LIN {X 0,Y 123.442,Z 476.669,A -85,B 0,C 180,E1 -28629.835,E2 -28629.835} C_VEL
LIN {X 0,Y 123.131,Z 478.566,A -85,B 0,C 180,E1 -28633.994,E2 -28633.994} C_VEL
LIN {X 0,Y 122.926,Z 480.125,A -85,B 0,C 180,E1 -28636.611,E2 -28636.611} C_VEL
LIN {X 0,Y 122.223,Z 482.877,A -85,B 0,C 180,E1 -28640.183,E2 -28640.183} C_VEL
LIN {X 0,Y 121.163,Z 486.4,A -85,B 0,C 180,E1 -28643.956,E2 -28643.956} C_VEL
LIN {X 0,Y 120.084,Z 488.681,A -85,B 0,C 180,E1 -28645.839,E2 -28645.839} C_VEL
LIN {X 0,Y 110.646,Z 498.011,A -85,B 0,C 180,E1 -28649.147,E2 -28649.147} C_VEL
LIN {X 0,Y 100.856,Z 506.281,A -85,B 0,C 180,E1 -28653.259,E2 -28653.259} C_VEL
LIN {X 0,Y 92.106,Z 512.776,A -85,B 0,C 180,E1 -28658.074,E2 -28658.074} C_VEL
LIN {X 0,Y 83.54,Z 518.436,A -85,B 0,C 180,E1 -28664.35,E2 -28664.35} C_VEL
LIN {X 0,Y 75.32,Z 523.224,A -85,B 0,C 180,E1 -28672.663,E2 -28672.663} C_VEL
LIN {X 0,Y 68.671,Z 526.759,A -85,B 0,C 180,E1 -28683.323,E2 -28683.323} C_VEL
LIN {X 0,Y 66.155,Z 527.832,A -85,B 0,C 180,E1 -28687.77,E2 -28687.77} C_VEL
LIN {X 0,Y 61.137,Z 529.24,A -85,B 0,C 180,E1 -28695.36,E2 -28695.36} C_VEL
LIN {X 0,Y 57.636,Z 529.91,A -85,B 0,C 180,E1 -28702.265,E2 -28702.265} C_VEL
LIN {X 0,Y 56.173,Z 530.076,A -85,B 0,C 180,E1 -28708.082,E2 -28708.082} C_VEL
LIN {X 0,Y 56.026,Z 530.057,A -85,B 0,C 180,E1 -28710.105,E2 -28710.105} C_VEL
LIN {X 0,Y 57.314,Z 529.481,A -85,B 0,C 180,E1 -28724.197,E2 -28724.197} C_VEL
LIN {X 0,Y 61.277,Z 527.703,A -85,B 0,C 180,E1 -28737.309,E2 -28737.309} C_VEL
LIN {X 0,Y 67.813,Z 524.66,A -85,B 0,C 180,E1 -28748.451,E2 -28748.451} C_VEL
LIN {X 0,Y 73.975,Z 521.492,A -85,B 0,C 180,E1 -28755.443,E2 -28755.443} C_VEL
LIN {X 0,Y 83.706,Z 515.997,A -85,B 0,C 180,E1 -28762.905,E2 -28762.905} C_VEL
LIN {X 0,Y 91.522,Z 510.885,A -85,B 0,C 180,E1 -28767.641,E2 -28767.641} C_VEL
LIN {X 0,Y 101.389,Z 503.57,A -85,B 0,C 180,E1 -28772.105,E2 -28772.105} C_VEL
LIN {X 0,Y 111.81,Z 494.625,A -85,B 0,C 180,E1 -28775.704,E2 -28775.704} C_VEL
LIN {X 0,Y 114.82,Z 491.688,A -85,B 0,C 180,E1 -28776.656,E2 -28776.656} C_VEL
LIN {X 0,Y 115.99,Z 490.149,A -85,B 0,C 180,E1 -28777.717,E2 -28777.717} C_VEL
LIN {X 0,Y 117.045,Z 487.526,A -85,B 0,C 180,E1 -28780.715,E2 -28780.715} C_VEL
LIN {X 0,Y 117.659,Z 485.914,A -85,B 0,C 180,E1 -28782.887,E2 -28782.887} C_VEL
LIN {X 0,Y 118.148,Z 483.965,A -85,B 0,C 180,E1 -28786.234,E2 -28786.234} C_VEL
LIN {X 0,Y 118.549,Z 482.415,A -85,B 0,C 180,E1 -28789.755,E2 -28789.755} C_VEL
LIN {X 0,Y 118.914,Z 481.354,A -85,B 0,C 180,E1 -28793.211,E2 -28793.211} C_VEL
LIN {X 0,Y 119.159,Z 480.799,A -85,B 0,C 180,E1 -28796.618,E2 -28796.618} C_VEL
LIN {X 0,Y 119.149,Z 480.971,A -85,B 0,C 180,E1 -28799.999,E2 -28799.999} C_VEL
LIN {X 0,Y 118.814,Z 481.957,A -85,B 0,C 180,E1 -28803.39,E2 -28803.39} C_VEL
LIN {X 0,Y 118.391,Z 483.416,A -85,B 0,C 180,E1 -28806.818,E2 -28806.818} C_VEL
LIN {X 0,Y 117.865,Z 485.41,A -85,B 0,C 180,E1 -28810.304,E2 -28810.304} C_VEL
LIN {X 0,Y 117.082,Z 488.121,A -85,B 0,C 180,E1 -28813.892,E2 -28813.892} C_VEL
LIN {X 0,Y 115.532,Z 492.582,A -85,B 0,C 180,E1 -28818.794,E2 -28818.794} C_VEL
LIN {X 0,Y 115.01,Z 493.547,A -85,B 0,C 180,E1 -28819.533,E2 -28819.533} C_VEL
LIN {X 0,Y 104.738,Z 503.117,A -85,B 0,C 180,E1 -28822.683,E2 -28822.683} C_VEL
LIN {X 0,Y 94.468,Z 511.413,A -85,B 0,C 180,E1 -28826.778,E2 -28826.778} C_VEL
LIN {X 0,Y 83.489,Z 519.074,A -85,B 0,C 180,E1 -28832.669,E2 -28832.669} C_VEL
LIN {X 0,Y 73.567,Z 525.093,A -85,B 0,C 180,E1 -28840.158,E2 -28840.158} C_VEL
LIN {X 0,Y 65.334,Z 529.662,A -85,B 0,C 180,E1 -28849.801,E2 -28849.801} C_VEL
LIN {X 0,Y 59.215,Z 532.878,A -85,B 0,C 180,E1 -28861.656,E2 -28861.656} C_VEL
LIN {X 0,Y 55.998,Z 534.817,A -85,B 0,C 180,E1 -28875.462,E2 -28875.462} C_VEL
LIN {X 0,Y 55.744,Z 535.501,A -85,B 0,C 180,E1 -28889.999,E2 -28889.999} C_VEL
LIN {X 0,Y 55.999,Z 534.796,A -85,B 0,C 180,E1 -28904.536,E2 -28904.536} C_VEL
LIN {X 0,Y 59.195,Z 532.826,A -85,B 0,C 180,E1 -28918.353,E2 -28918.353} C_VEL
LIN {X 0,Y 65.247,Z 529.584,A -85,B 0,C 180,E1 -28930.261,E2 -28930.261} C_VEL
LIN {X 0,Y 73.545,Z 524.995,A -85,B 0,C 180,E1 -28939.861,E2 -28939.861} C_VEL
LIN {X 0,Y 83.473,Z 518.938,A -85,B 0,C 180,E1 -28947.347,E2 -28947.347} C_VEL
LIN {X 0,Y 94.427,Z 511.231,A -85,B 0,C 180,E1 -28953.27,E2 -28953.27} C_VEL
LIN {X 0,Y 104.716,Z 502.903,A -85,B 0,C 180,E1 -28957.344,E2 -28957.344} C_VEL
LIN {X 0,Y 114.943,Z 493.322,A -85,B 0,C 180,E1 -28960.492,E2 -28960.492} C_VEL
LIN {X 0,Y 115.872,Z 491.229,A -85,B 0,C 180,E1 -28962.347,E2 -28962.347} C_VEL
LIN {X 0,Y 117.35,Z 486.686,A -85,B 0,C 180,E1 -28967.619,E2 -28967.619} C_VEL
LIN {X 0,Y 117.773,Z 485.194,A -85,B 0,C 180,E1 -28969.688,E2 -28969.688} C_VEL
LIN {X 0,Y 118.264,Z 483.229,A -85,B 0,C 180,E1 -28973.175,E2 -28973.175} C_VEL
LIN {X 0,Y 118.678,Z 481.763,A -85,B 0,C 180,E1 -28976.606,E2 -28976.606} C_VEL
LIN {X 0,Y 119.054,Z 480.719,A -85,B 0,C 180,E1 -28980.001,E2 -28980.001} C_VEL
LIN {X 0,Y 119.069,Z 480.536,A -85,B 0,C 180,E1 -28983.384,E2 -28983.384} C_VEL
LIN {X 0,Y 118.726,Z 481.294,A -85,B 0,C 180,E1 -28987.438,E2 -28987.438} C_VEL
LIN {X 0,Y 118.472,Z 482.151,A -85,B 0,C 180,E1 -28990.252,E2 -28990.252} C_VEL
LIN {X 0,Y 118.083,Z 483.683,A -85,B 0,C 180,E1 -28993.773,E2 -28993.773} C_VEL
LIN {X 0,Y 117.525,Z 485.84,A -85,B 0,C 180,E1 -28997.398,E2 -28997.398} C_VEL
LIN {X 0,Y 115.975,Z 489.809,A -85,B 0,C 180,E1 -29002.234,E2 -29002.234} C_VEL
LIN {X 0,Y 114.863,Z 491.379,A -85,B 0,C 180,E1 -29003.395,E2 -29003.395} C_VEL
LIN {X 0,Y 104.387,Z 500.893,A -85,B 0,C 180,E1 -29006.864,E2 -29006.864} C_VEL
LIN {X 0,Y 94.332,Z 508.689,A -85,B 0,C 180,E1 -29011.043,E2 -29011.043} C_VEL
LIN {X 0,Y 86.254,Z 514.244,A -85,B 0,C 180,E1 -29015.432,E2 -29015.432} C_VEL
LIN {X 0,Y 78.74,Z 518.785,A -85,B 0,C 180,E1 -29020.653,E2 -29020.653} C_VEL
LIN {X 0,Y 69.786,Z 523.572,A -85,B 0,C 180,E1 -29029.111,E2 -29029.111} C_VEL
LIN {X 0,Y 62.167,Z 527.216,A -85,B 0,C 180,E1 -29040.869,E2 -29040.869} C_VEL
LIN {X 0,Y 58.97,Z 528.699,A -85,B 0,C 180,E1 -29049.052,E2 -29049.052} C_VEL
LIN {X 0,Y 56.296,Z 529.907,A -85,B 0,C 180,E1 -29062.829,E2 -29062.829} C_VEL
LIN {X 0,Y 56.026,Z 530.057,A -85,B 0,C 180,E1 -29070.105,E2 -29070.105} C_VEL
LIN {X 0,Y 55.496,Z 529.985,A -85,B 0,C 180,E1 -29076.152,E2 -29076.152} C_VEL
LIN {X 0,Y 54.053,Z 529.556,A -85,B 0,C 180,E1 -29086.427,E2 -29086.427} C_VEL
LIN {X 0,Y 53.917,Z 528.842,A -85,B 0,C 180,E1 -29094.874,E2 -29094.874} C_VEL
LIN {X 0,Y 55.248,Z 528.005,A -85,B 0,C 180,E1 -29100.892,E2 -29100.892} C_VEL
LIN {X 0,Y 56.05,Z 527.625,A -85,B 0,C 180,E1 -29102.721,E2 -29102.721} C_VEL
LIN {X 0,Y 64.524,Z 524.032,A -85,B 0,C 180,E1 -29115.073,E2 -29115.073} C_VEL
LIN {X 0,Y 74.271,Z 519.28,A -85,B 0,C 180,E1 -29123.546,E2 -29123.546} C_VEL
LIN {X 0,Y 84.459,Z 513.418,A -85,B 0,C 180,E1 -29129.824,E2 -29129.824} C_VEL
LIN {X 0,Y 95.251,Z 506.136,A -85,B 0,C 180,E1 -29134.672,E2 -29134.672} C_VEL
LIN {X 0,Y 105.982,Z 497.686,A -85,B 0,C 180,E1 -29138.187,E2 -29138.187} C_VEL
LIN {X 0,Y 110.875,Z 493.225,A -85,B 0,C 180,E1 -29139.785,E2 -29139.785} C_VEL
LIN {X 0,Y 112.206,Z 490.669,A -85,B 0,C 180,E1 -29143.22,E2 -29143.22} C_VEL
LIN {X 0,Y 112.67,Z 489.356,A -85,B 0,C 180,E1 -29145.551,E2 -29145.551} C_VEL
LIN {X 0,Y 113.3,Z 487.678,A -85,B 0,C 180,E1 -29149.275,E2 -29149.275} C_VEL
LIN {X 0,Y 113.819,Z 486.542,A -85,B 0,C 180,E1 -29152.906,E2 -29152.906} C_VEL
LIN {X 0,Y 114.16,Z 485.933,A -85,B 0,C 180,E1 -29156.47,E2 -29156.47} C_VEL
LIN {X 0,Y 114.154,Z 486.101,A -85,B 0,C 180,E1 -29159.999,E2 -29159.999} C_VEL
LIN {X 0,Y 113.684,Z 487.173,A -85,B 0,C 180,E1 -29163.544,E2 -29163.544} C_VEL
LIN {X 0,Y 113.087,Z 488.722,A -85,B 0,C 180,E1 -29167.139,E2 -29167.139} C_VEL
LIN {X 0,Y 112.312,Z 490.85,A -85,B 0,C 180,E1 -29170.819,E2 -29170.819} C_VEL
LIN {X 0,Y 111.093,Z 493.787,A -85,B 0,C 180,E1 -29174.657,E2 -29174.657} C_VEL
LIN {X 0,Y 110.108,Z 495.718,A -85,B 0,C 180,E1 -29176.776,E2 -29176.776} C_VEL
LIN {X 0,Y 99.067,Z 505.251,A -85,B 0,C 180,E1 -29179.949,E2 -29179.949} C_VEL
LIN {X 0,Y 89.974,Z 512.085,A -85,B 0,C 180,E1 -29183.39,E2 -29183.39} C_VEL
LIN {X 0,Y 79.849,Z 518.722,A -85,B 0,C 180,E1 -29188.336,E2 -29188.336} C_VEL
LIN {X 0,Y 69.139,Z 524.742,A -85,B 0,C 180,E1 -29195.589,E2 -29195.589} C_VEL
LIN {X 0,Y 60.013,Z 529.312,A -85,B 0,C 180,E1 -29205.359,E2 -29205.359} C_VEL
LIN {X 0,Y 53.023,Z 532.53,A -85,B 0,C 180,E1 -29217.981,E2 -29217.981} C_VEL
LIN {X 0,Y 49.106,Z 534.47,A -85,B 0,C 180,E1 -29233.366,E2 -29233.366} C_VEL
LIN {X 0,Y 48.634,Z 535.155,A -85,B 0,C 180,E1 -29249.999,E2 -29249.999} C_VEL
LIN {X 0,Y 49.106,Z 534.448,A -85,B 0,C 180,E1 -29266.632,E2 -29266.632} C_VEL
LIN {X 0,Y 53,Z 532.477,A -85,B 0,C 180,E1 -29282.033,E2 -29282.033} C_VEL
LIN {X 0,Y 59.933,Z 529.232,A -85,B 0,C 180,E1 -29294.715,E2 -29294.715} C_VEL
LIN {X 0,Y 69.125,Z 524.641,A -85,B 0,C 180,E1 -29304.426,E2 -29304.426} C_VEL
LIN {X 0,Y 79.832,Z 518.584,A -85,B 0,C 180,E1 -29311.684,E2 -29311.684} C_VEL
LIN {X 0,Y 91.413,Z 510.868,A -85,B 0,C 180,E1 -29317.306,E2 -29317.306} C_VEL
LIN {X 0,Y 102.167,Z 502.533,A -85,B 0,C 180,E1 -29321.059,E2 -29321.059} C_VEL
LIN {X 0,Y 110.092,Z 495.463,A -85,B 0,C 180,E1 -29323.248,E2 -29323.248} C_VEL
LIN {X 0,Y 111.044,Z 493.576,A -85,B 0,C 180,E1 -29325.336,E2 -29325.336} C_VEL
LIN {X 0,Y 112.232,Z 490.64,A -85,B 0,C 180,E1 -29329.173,E2 -29329.173} C_VEL
LIN {X 0,Y 113.147,Z 488.13,A -85,B 0,C 180,E1 -29333.629,E2 -29333.629} C_VEL
LIN {X 0,Y 113.558,Z 486.983,A -85,B 0,C 180,E1 -29336.452,E2 -29336.452} C_VEL
LIN {X 0,Y 114.055,Z 485.873,A -85,B 0,C 180,E1 -29340.001,E2 -29340.001} C_VEL
LIN {X 0,Y 114.08,Z 485.68,A -85,B 0,C 180,E1 -29343.533,E2 -29343.533} C_VEL
LIN {X 0,Y 113.59,Z 486.589,A -85,B 0,C 180,E1 -29348.132,E2 -29348.132} C_VEL
LIN {X 0,Y 113.231,Z 487.427,A -85,B 0,C 180,E1 -29350.732,E2 -29350.732} C_VEL
LIN {X 0,Y 112.605,Z 489.096,A -85,B 0,C 180,E1 -29354.458,E2 -29354.458} C_VEL
LIN {X 0,Y 112.16,Z 490.362,A -85,B 0,C 180,E1 -29356.693,E2 -29356.693} C_VEL
LIN {X 0,Y 110.825,Z 492.996,A -85,B 0,C 180,E1 -29360.279,E2 -29360.279} C_VEL
LIN {X 0,Y 107.557,Z 496.07,A -85,B 0,C 180,E1 -29361.389,E2 -29361.389} C_VEL
LIN {X 0,Y 96.809,Z 504.795,A -85,B 0,C 180,E1 -29364.844,E2 -29364.844} C_VEL
LIN {X 0,Y 86.811,Z 511.771,A -85,B 0,C 180,E1 -29369.062,E2 -29369.062} C_VEL
LIN {X 0,Y 76.956,Z 517.733,A -85,B 0,C 180,E1 -29374.723,E2 -29374.723} C_VEL
LIN {X 0,Y 66.816,Z 522.882,A -85,B 0,C 180,E1 -29382.584,E2 -29382.584} C_VEL
LIN {X 0,Y 58.485,Z 526.608,A -85,B 0,C 180,E1 -29393.071,E2 -29393.071} C_VEL
LIN {X 0,Y 52.417,Z 529.044,A -85,B 0,C 180,E1 -29406.283,E2 -29406.283} C_VEL
LIN {X 0,Y 49.28,Z 530.252,A -85,B 0,C 180,E1 -29421.802,E2 -29421.802} C_VEL
LIN {X 0,Y 48.949,Z 530.404,A -85,B 0,C 180,E1 -29430.001,E2 -29430.001} C_VEL
LIN {X 0,Y 50.461,Z 529.826,A -85,B 0,C 180,E1 -29446.175,E2 -29446.175} C_VEL
LIN {X 0,Y 55.071,Z 528.048,A -85,B 0,C 180,E1 -29460.696,E2 -29460.696} C_VEL
LIN {X 0,Y 56.05,Z 527.625,A -85,B 0,C 180,E1 -29462.721,E2 -29462.721} C_VEL
LIN {X 0,Y 58.351,Z 526.555,A -85,B 0,C 180,E1 -29468.046,E2 -29468.046} C_VEL
LIN {X 0,Y 61.578,Z 524.441,A -85,B 0,C 180,E1 -29476.786,E2 -29476.786} C_VEL
LIN {X 0,Y 65.945,Z 521.835,A -85,B 0,C 180,E1 -29484.444,E2 -29484.444} C_VEL
LIN {X 0,Y 69.769,Z 519.876,A -85,B 0,C 180,E1 -29487.874,E2 -29487.874} C_VEL
LIN {X 0,Y 78.831,Z 515.114,A -85,B 0,C 180,E1 -29493.067,E2 -29493.067} C_VEL
LIN {X 0,Y 89.345,Z 508.618,A -85,B 0,C 180,E1 -29497.561,E2 -29497.561} C_VEL
LIN {X 0,Y 100.366,Z 500.648,A -85,B 0,C 180,E1 -29500.967,E2 -29500.967} C_VEL
LIN {X 0,Y 106.067,Z 495.905,A -85,B 0,C 180,E1 -29502.611,E2 -29502.611} C_VEL
LIN {X 0,Y 106.883,Z 494.538,A -85,B 0,C 180,E1 -29504.75,E2 -29504.75} C_VEL
LIN {X 0,Y 107.731,Z 492.77,A -85,B 0,C 180,E1 -29508.713,E2 -29508.713} C_VEL
LIN {X 0,Y 108.493,Z 491.5,A -85,B 0,C 180,E1 -29512.555,E2 -29512.555} C_VEL
LIN {X 0,Y 108.936,Z 490.843,A -85,B 0,C 180,E1 -29516.3,E2 -29516.3} C_VEL
LIN {X 0,Y 108.916,Z 491.025,A -85,B 0,C 180,E1 -29519.999,E2 -29519.999} C_VEL
LIN {X 0,Y 108.316,Z 492.16,A -85,B 0,C 180,E1 -29523.72,E2 -29523.72} C_VEL
LIN {X 0,Y 107.558,Z 493.767,A -85,B 0,C 180,E1 -29527.508,E2 -29527.508} C_VEL
LIN {X 0,Y 106.414,Z 496.104,A -85,B 0,C 180,E1 -29531.427,E2 -29531.427} C_VEL
LIN {X 0,Y 104.974,Z 498.293,A -85,B 0,C 180,E1 -29533.882,E2 -29533.882} C_VEL
LIN {X 0,Y 93.645,Z 507.308,A -85,B 0,C 180,E1 -29536.883,E2 -29536.883} C_VEL
LIN {X 0,Y 82.737,Z 514.756,A -85,B 0,C 180,E1 -29540.869,E2 -29540.869} C_VEL
LIN {X 0,Y 70.811,Z 521.57,A -85,B 0,C 180,E1 -29546.713,E2 -29546.713} C_VEL
LIN {X 0,Y 59.957,Z 526.851,A -85,B 0,C 180,E1 -29554.862,E2 -29554.862} C_VEL
LIN {X 0,Y 50.779,Z 530.735,A -85,B 0,C 180,E1 -29566.208,E2 -29566.208} C_VEL
LIN {X 0,Y 44.196,Z 533.307,A -85,B 0,C 180,E1 -29581.506,E2 -29581.506} C_VEL
LIN {X 0,Y 41.413,Z 534.624,A -85,B 0,C 180,E1 -29600.228,E2 -29600.228} C_VEL
LIN {X 0,Y 41.523,Z 534.809,A -85,B 0,C 180,E1 -29609.999,E2 -29609.999} C_VEL
LIN {X 0,Y 42.294,Z 534.099,A -85,B 0,C 180,E1 -29629.41,E2 -29629.41} C_VEL
LIN {X 0,Y 47.059,Z 532.127,A -85,B 0,C 180,E1 -29646.681,E2 -29646.681} C_VEL
LIN {X 0,Y 56.01,Z 528.494,A -85,B 0,C 180,E1 -29661.144,E2 -29661.144} C_VEL
LIN {X 0,Y 65.214,Z 524.29,A -85,B 0,C 180,E1 -29669.557,E2 -29669.557} C_VEL
LIN {X 0,Y 76.678,Z 518.228,A -85,B 0,C 180,E1 -29676.428,E2 -29676.428} C_VEL
LIN {X 0,Y 88.885,Z 510.505,A -85,B 0,C 180,E1 -29681.589,E2 -29681.589} C_VEL
LIN {X 0,Y 100.07,Z 502.162,A -85,B 0,C 180,E1 -29684.944,E2 -29684.944} C_VEL
LIN {X 0,Y 104.963,Z 498.059,A -85,B 0,C 180,E1 -29686.138,E2 -29686.138} C_VEL
LIN {X 0,Y 106.311,Z 495.933,A -85,B 0,C 180,E1 -29688.562,E2 -29688.562} C_VEL
LIN {X 0,Y 107.467,Z 493.58,A -85,B 0,C 180,E1 -29692.485,E2 -29692.485} C_VEL
LIN {X 0,Y 108.206,Z 491.973,A -85,B 0,C 180,E1 -29696.277,E2 -29696.277} C_VEL
LIN {X 0,Y 108.816,Z 490.819,A -85,B 0,C 180,E1 -29700.001,E2 -29700.001} C_VEL
LIN {X 0,Y 108.867,Z 490.603,A -85,B 0,C 180,E1 -29703.702,E2 -29703.702} C_VEL
LIN {X 0,Y 108.422,Z 491.268,A -85,B 0,C 180,E1 -29707.45,E2 -29707.45} C_VEL
LIN {X 0,Y 107.61,Z 492.646,A -85,B 0,C 180,E1 -29711.58,E2 -29711.58} C_VEL
LIN {X 0,Y 106.822,Z 494.3,A -85,B 0,C 180,E1 -29715.259,E2 -29715.259} C_VEL
LIN {X 0,Y 106.018,Z 495.674,A -85,B 0,C 180,E1 -29717.388,E2 -29717.388} C_VEL
LIN {X 0,Y 102.001,Z 499.115,A -85,B 0,C 180,E1 -29718.667,E2 -29718.667} C_VEL
LIN {X 0,Y 90.938,Z 507.36,A -85,B 0,C 180,E1 -29721.966,E2 -29721.966} C_VEL
LIN {X 0,Y 81.2,Z 513.552,A -85,B 0,C 180,E1 -29725.867,E2 -29725.867} C_VEL
LIN {X 0,Y 70.311,Z 519.484,A -85,B 0,C 180,E1 -29731.83,E2 -29731.83} C_VEL
LIN {X 0,Y 59.76,Z 524.267,A -85,B 0,C 180,E1 -29740.145,E2 -29740.145} C_VEL
LIN {X 0,Y 52.988,Z 526.954,A -85,B 0,C 180,E1 -29748.458,E2 -29748.458} C_VEL
LIN {X 0,Y 46.008,Z 529.389,A -85,B 0,C 180,E1 -29762.725,E2 -29762.725} C_VEL
LIN {X 0,Y 42.284,Z 530.597,A -85,B 0,C 180,E1 -29780.433,E2 -29780.433} C_VEL
LIN {X 0,Y 41.858,Z 530.749,A -85,B 0,C 180,E1 -29790.001,E2 -29790.001} C_VEL
LIN {X 0,Y 43.704,Z 530.17,A -85,B 0,C 180,E1 -29808.762,E2 -29808.762} C_VEL
LIN {X 0,Y 49.089,Z 528.393,A -85,B 0,C 180,E1 -29824.939,E2 -29824.939} C_VEL
LIN {X 0,Y 57.355,Z 525.35,A -85,B 0,C 180,E1 -29837.326,E2 -29837.326} C_VEL
LIN {X 0,Y 64.81,Z 522.185,A -85,B 0,C 180,E1 -29844.421,E2 -29844.421} C_VEL
LIN {X 0,Y 69.769,Z 519.876,A -85,B 0,C 180,E1 -29847.874,E2 -29847.874} C_VEL
LIN {X 0,Y 73.744,Z 517.773,A -85,B 0,C 180,E1 -29850.933,E2 -29850.933} C_VEL
LIN {X 0,Y 79.475,Z 514.137,A -85,B 0,C 180,E1 -29856.351,E2 -29856.351} C_VEL
LIN {X 0,Y 85.555,Z 509.963,A -85,B 0,C 180,E1 -29860.962,E2 -29860.962} C_VEL
LIN {X 0,Y 89.849,Z 507.018,A -85,B 0,C 180,E1 -29862.783,E2 -29862.783} C_VEL
LIN {X 0,Y 99.92,Z 499.756,A -85,B 0,C 180,E1 -29865.27,E2 -29865.27} C_VEL
LIN {X 0,Y 101.388,Z 498.453,A -85,B 0,C 180,E1 -29866.041,E2 -29866.041} C_VEL
LIN {X 0,Y 102.833,Z 496.309,A -85,B 0,C 180,E1 -29872.143,E2 -29872.143} C_VEL
LIN {X 0,Y 103.477,Z 495.538,A -85,B 0,C 180,E1 -29876.105,E2 -29876.105} C_VEL
LIN {X 0,Y 103.441,Z 495.733,A -85,B 0,C 180,E1 -29879.999,E2 -29879.999} C_VEL
LIN {X 0,Y 102.684,Z 496.938,A -85,B 0,C 180,E1 -29883.924,E2 -29883.924} C_VEL
LIN {X 0,Y 101.293,Z 499.271,A -85,B 0,C 180,E1 -29889.07,E2 -29889.07} C_VEL
LIN {X 0,Y 100.135,Z 500.664,A -85,B 0,C 180,E1 -29890.701,E2 -29890.701} C_VEL
LIN {X 0,Y 88.537,Z 509.216,A -85,B 0,C 180,E1 -29893.489,E2 -29893.489} C_VEL
LIN {X 0,Y 77.275,Z 516.245,A -85,B 0,C 180,E1 -29897.26,E2 -29897.26} C_VEL
LIN {X 0,Y 64.854,Z 522.675,A -85,B 0,C 180,E1 -29902.907,E2 -29902.907} C_VEL
LIN {X 0,Y 56.15,Z 526.501,A -85,B 0,C 180,E1 -29908.816,E2 -29908.816} C_VEL
LIN {X 0,Y 45.865,Z 530.387,A -85,B 0,C 180,E1 -29919.988,E2 -29919.988} C_VEL
LIN {X 0,Y 38.041,Z 532.958,A -85,B 0,C 180,E1 -29936.34,E2 -29936.34} C_VEL
LIN {X 0,Y 34.386,Z 534.276,A -85,B 0,C 180,E1 -29958.205,E2 -29958.205} C_VEL
LIN {X 0,Y 34.404,Z 534.462,A -85,B 0,C 180,E1 -29969.999,E2 -29969.999} C_VEL
LIN {X 0,Y 35.629,Z 533.751,A -85,B 0,C 180,E1 -29993.235,E2 -29993.235} C_VEL
LIN {X 0,Y 41.521,Z 531.777,A -85,B 0,C 180,E1 -30012.613,E2 -30012.613} C_VEL
LIN {X 0,Y 51.108,Z 528.395,A -85,B 0,C 180,E1 -30026.631,E2 -30026.631} C_VEL
LIN {X 0,Y 61.881,Z 523.938,A -85,B 0,C 180,E1 -30035.309,E2 -30035.309} C_VEL
LIN {X 0,Y 74.095,Z 517.873,A -85,B 0,C 180,E1 -30041.533,E2 -30041.533} C_VEL
LIN {X 0,Y 86.885,Z 510.142,A -85,B 0,C 180,E1 -30046.086,E2 -30046.086} C_VEL
LIN {X 0,Y 98.45,Z 501.79,A -85,B 0,C 180,E1 -30048.982,E2 -30048.982} C_VEL
LIN {X 0,Y 100.125,Z 500.423,A -85,B 0,C 180,E1 -30049.324,E2 -30049.324} C_VEL
LIN {X 0,Y 101.578,Z 498.488,A -85,B 0,C 180,E1 -30052.047,E2 -30052.047} C_VEL
LIN {X 0,Y 102.585,Z 496.759,A -85,B 0,C 180,E1 -30056.072,E2 -30056.072} C_VEL
LIN {X 0,Y 103.341,Z 495.545,A -85,B 0,C 180,E1 -30060.001,E2 -30060.001} C_VEL
LIN {X 0,Y 103.413,Z 495.315,A -85,B 0,C 180,E1 -30063.898,E2 -30063.898} C_VEL
LIN {X 0,Y 102.794,Z 496.074,A -85,B 0,C 180,E1 -30067.86,E2 -30067.86} C_VEL
LIN {X 0,Y 101.356,Z 498.195,A -85,B 0,C 180,E1 -30073.889,E2 -30073.889} C_VEL
LIN {X 0,Y 99.953,Z 499.485,A -85,B 0,C 180,E1 -30074.804,E2 -30074.804} C_VEL
LIN {X 0,Y 88.524,Z 507.721,A -85,B 0,C 180,E1 -30077.694,E2 -30077.694} C_VEL
LIN {X 0,Y 77.848,Z 514.202,A -85,B 0,C 180,E1 -30081.395,E2 -30081.395} C_VEL
LIN {X 0,Y 66.84,Z 519.834,A -85,B 0,C 180,E1 -30086.653,E2 -30086.653} C_VEL
LIN {X 0,Y 55.446,Z 524.615,A -85,B 0,C 180,E1 -30094.523,E2 -30094.523} C_VEL
LIN {X 0,Y 47.901,Z 527.3,A -85,B 0,C 180,E1 -30102.812,E2 -30102.812} C_VEL
LIN {X 0,Y 39.825,Z 529.735,A -85,B 0,C 180,E1 -30118.035,E2 -30118.035} C_VEL
LIN {X 0,Y 35.308,Z 530.942,A -85,B 0,C 180,E1 -30138.52,E2 -30138.52} C_VEL
LIN {X 0,Y 34.777,Z 531.094,A -85,B 0,C 180,E1 -30150.001,E2 -30150.001} C_VEL
LIN {X 0,Y 37.05,Z 530.516,A -85,B 0,C 180,E1 -30172.297,E2 -30172.297} C_VEL
LIN {X 0,Y 43.453,Z 528.738,A -85,B 0,C 180,E1 -30190.313,E2 -30190.313} C_VEL
LIN {X 0,Y 52.785,Z 525.696,A -85,B 0,C 180,E1 -30203.023,E2 -30203.023} C_VEL
LIN {X 0,Y 60.958,Z 522.531,A -85,B 0,C 180,E1 -30209.85,E2 -30209.85} C_VEL
LIN {X 0,Y 72.839,Z 517.047,A -85,B 0,C 180,E1 -30216.44,E2 -30216.44} C_VEL
LIN {X 0,Y 82.109,Z 511.939,A -85,B 0,C 180,E1 -30220.312,E2 -30220.312} C_VEL
LIN {X 0,Y 89.849,Z 507.018,A -85,B 0,C 180,E1 -30222.783,E2 -30222.783} C_VEL
LIN {X 0,Y 92.101,Z 505.395,A -85,B 0,C 180,E1 -30223.881,E2 -30223.881} C_VEL
LIN {X 0,Y 94.335,Z 503.478,A -85,B 0,C 180,E1 -30226.133,E2 -30226.133} C_VEL
LIN {X 0,Y 95.937,Z 501.855,A -85,B 0,C 180,E1 -30229.234,E2 -30229.234} C_VEL
LIN {X 0,Y 96.981,Z 500.764,A -85,B 0,C 180,E1 -30232.579,E2 -30232.579} C_VEL
LIN {X 0,Y 97.378,Z 500.354,A -85,B 0,C 180,E1 -30234.27,E2 -30234.27} C_VEL
LIN {X 0,Y 97.772,Z 500.02,A -85,B 0,C 180,E1 -30235.877,E2 -30235.877} C_VEL
LIN {X 0,Y 97.74,Z 500.212,A -85,B 0,C 180,E1 -30239.999,E2 -30239.999} C_VEL
LIN {X 0,Y 96.286,Z 502.168,A -85,B 0,C 180,E1 -30245.848,E2 -30245.848} C_VEL
LIN {X 0,Y 94.974,Z 503.397,A -85,B 0,C 180,E1 -30247.324,E2 -30247.324} C_VEL
LIN {X 0,Y 82.51,Z 511.782,A -85,B 0,C 180,E1 -30249.993,E2 -30249.993} C_VEL
LIN {X 0,Y 72.155,Z 517.665,A -85,B 0,C 180,E1 -30253.086,E2 -30253.086} C_VEL
LIN {X 0,Y 59.247,Z 523.693,A -85,B 0,C 180,E1 -30258.379,E2 -30258.379} C_VEL
LIN {X 0,Y 47.164,Z 528.265,A -85,B 0,C 180,E1 -30266.606,E2 -30266.606} C_VEL
LIN {X 0,Y 36.59,Z 531.484,A -85,B 0,C 180,E1 -30279.797,E2 -30279.797} C_VEL
LIN {X 0,Y 29.173,Z 533.425,A -85,B 0,C 180,E1 -30301.194,E2 -30301.194} C_VEL
LIN {X 0,Y 27.276,Z 534.115,A -85,B 0,C 180,E1 -30329.998,E2 -30329.998} C_VEL
LIN {X 0,Y 29.168,Z 533.402,A -85,B 0,C 180,E1 -30358.808,E2 -30358.808} C_VEL
LIN {X 0,Y 36.564,Z 531.428,A -85,B 0,C 180,E1 -30380.248,E2 -30380.248} C_VEL
LIN {X 0,Y 47.11,Z 528.18,A -85,B 0,C 180,E1 -30393.521,E2 -30393.521} C_VEL
LIN {X 0,Y 59.242,Z 523.586,A -85,B 0,C 180,E1 -30401.631,E2 -30401.631} C_VEL
LIN {X 0,Y 72.141,Z 517.518,A -85,B 0,C 180,E1 -30406.956,E2 -30406.956} C_VEL
LIN {X 0,Y 83.47,Z 510.996,A -85,B 0,C 180,E1 -30410.306,E2 -30410.306} C_VEL
LIN {X 0,Y 94.886,Z 503.227,A -85,B 0,C 180,E1 -30412.706,E2 -30412.706} C_VEL
LIN {X 0,Y 96.216,Z 501.989,A -85,B 0,C 180,E1 -30414.176,E2 -30414.176} C_VEL
LIN {X 0,Y 97.634,Z 500.043,A -85,B 0,C 180,E1 -30420.001,E2 -30420.001} C_VEL
LIN {X 0,Y 97.718,Z 499.809,A -85,B 0,C 180,E1 -30424.125,E2 -30424.125} C_VEL
LIN {X 0,Y 96.881,Z 500.67,A -85,B 0,C 180,E1 -30428.343,E2 -30428.343} C_VEL
LIN {X 0,Y 96.463,Z 501.121,A -85,B 0,C 180,E1 -30429.863,E2 -30429.863} C_VEL
LIN {X 0,Y 95.238,Z 502.175,A -85,B 0,C 180,E1 -30431.386,E2 -30431.386} C_VEL
LIN {X 0,Y 83.319,Z 510.112,A -85,B 0,C 180,E1 -30434.064,E2 -30434.064} C_VEL
LIN {X 0,Y 70.315,Z 517.236,A -85,B 0,C 180,E1 -30438.283,E2 -30438.283} C_VEL
LIN {X 0,Y 57.743,Z 522.756,A -85,B 0,C 180,E1 -30444.101,E2 -30444.101} C_VEL
LIN {X 0,Y 48.875,Z 525.951,A -85,B 0,C 180,E1 -30450.371,E2 -30450.371} C_VEL
LIN {X 0,Y 38.352,Z 529.02,A -85,B 0,C 180,E1 -30462.863,E2 -30462.863} C_VEL
LIN {X 0,Y 30.618,Z 530.834,A -85,B 0,C 180,E1 -30482.674,E2 -30482.674} C_VEL
LIN {X 0,Y 27.698,Z 531.439,A -85,B 0,C 180,E1 -30510.002,E2 -30510.002} C_VEL
LIN {X 0,Y 30.613,Z 530.86,A -85,B 0,C 180,E1 -30537.334,E2 -30537.334} C_VEL
LIN {X 0,Y 38.317,Z 529.082,A -85,B 0,C 180,E1 -30557.197,E2 -30557.197} C_VEL
LIN {X 0,Y 48.832,Z 526.042,A -85,B 0,C 180,E1 -30569.719,E2 -30569.719} C_VEL
LIN {X 0,Y 60.819,Z 521.653,A -85,B 0,C 180,E1 -30577.588,E2 -30577.588} C_VEL
LIN {X 0,Y 70.291,Z 517.398,A -85,B 0,C 180,E1 -30581.782,E2 -30581.782} C_VEL
LIN {X 0,Y 79.997,Z 512.289,A -85,B 0,C 180,E1 -30585.107,E2 -30585.107} C_VEL
LIN {X 0,Y 91.616,Z 504.991,A -85,B 0,C 180,E1 -30587.985,E2 -30587.985} C_VEL
LIN {X 0,Y 95.284,Z 502.374,A -85,B 0,C 180,E1 -30588.676,E2 -30588.676} C_VEL
LIN {X 0,Y 96.497,Z 501.33,A -85,B 0,C 180,E1 -30590.173,E2 -30590.173} C_VEL
LIN {X 0,Y 97.378,Z 500.354,A -85,B 0,C 180,E1 -30594.27,E2 -30594.27} C_VEL
LIN {X 0,Y 97.034,Z 500.596,A -85,B 0,C 180,E1 -30595.506,E2 -30595.506} C_VEL
LIN {X 0,Y 95.028,Z 502.046,A -85,B 0,C 180,E1 -30597.237,E2 -30597.237} C_VEL
LIN {X 0,Y 92.2,Z 504.141,A -85,B 0,C 180,E1 -30599.422,E2 -30599.422} C_VEL
LIN {X 0,Y 91.694,Z 504.567,A -85,B 0,C 180,E1 -30600.351,E2 -30600.351} C_VEL
LIN {X 0,Y 91.222,Z 505.094,A -85,B 0,C 180,E1 -30602.205,E2 -30602.205} C_VEL
LIN {X 0,Y 89.856,Z 506.187,A -85,B 0,C 180,E1 -30603.625,E2 -30603.625} C_VEL
LIN {X 0,Y 77.713,Z 513.693,A -85,B 0,C 180,E1 -30605.843,E2 -30605.843} C_VEL
LIN {X 0,Y 64.083,Z 520.518,A -85,B 0,C 180,E1 -30609.231,E2 -30609.231} C_VEL
LIN {X 0,Y 50.808,Z 525.802,A -85,B 0,C 180,E1 -30614.465,E2 -30614.465} C_VEL
LIN {X 0,Y 38.257,Z 529.69,A -85,B 0,C 180,E1 -30623.284,E2 -30623.284} C_VEL
LIN {X 0,Y 27.278,Z 532.261,A -85,B 0,C 180,E1 -30639.379,E2 -30639.379} C_VEL
LIN {X 0,Y 20.61,Z 533.581,A -85,B 0,C 180,E1 -30670.06,E2 -30670.06} C_VEL
LIN {X 0,Y 20.169,Z 533.769,A -85,B 0,C 180,E1 -30689.998,E2 -30689.998} C_VEL
LIN {X 0,Y 23.141,Z 533.052,A -85,B 0,C 180,E1 -30727.399,E2 -30727.399} C_VEL
LIN {X 0,Y 32.451,Z 531.079,A -85,B 0,C 180,E1 -30750.028,E2 -30750.028} C_VEL
LIN {X 0,Y 44.375,Z 527.829,A -85,B 0,C 180,E1 -30761.854,E2 -30761.854} C_VEL
LIN {X 0,Y 57.38,Z 523.234,A -85,B 0,C 180,E1 -30768.477,E2 -30768.477} C_VEL
LIN {X 0,Y 70.866,Z 517.163,A -85,B 0,C 180,E1 -30772.627,E2 -30772.627} C_VEL
LIN {X 0,Y 81.632,Z 511.189,A -85,B 0,C 180,E1 -30775.062,E2 -30775.062} C_VEL
LIN {X 0,Y 89.825,Z 505.994,A -85,B 0,C 180,E1 -30776.424,E2 -30776.424} C_VEL
LIN {X 0,Y 91.181,Z 504.868,A -85,B 0,C 180,E1 -30778.013,E2 -30778.013} C_VEL
LIN {X 0,Y 91.707,Z 504.299,A -85,B 0,C 180,E1 -30780.001,E2 -30780.001} C_VEL
LIN {X 0,Y 91.685,Z 504.147,A -85,B 0,C 180,E1 -30784.793,E2 -30784.793} C_VEL
LIN {X 0,Y 91.333,Z 504.438,A -85,B 0,C 180,E1 -30786.407,E2 -30786.407} C_VEL
LIN {X 0,Y 90.046,Z 505.366,A -85,B 0,C 180,E1 -30787.739,E2 -30787.739} C_VEL
LIN {X 0,Y 78.486,Z 512.454,A -85,B 0,C 180,E1 -30789.938,E2 -30789.938} C_VEL
LIN {X 0,Y 65.103,Z 519.129,A -85,B 0,C 180,E1 -30793.695,E2 -30793.695} C_VEL
LIN {X 0,Y 51.981,Z 524.269,A -85,B 0,C 180,E1 -30798.842,E2 -30798.842} C_VEL
LIN {X 0,Y 39.627,Z 527.993,A -85,B 0,C 180,E1 -30807.532,E2 -30807.532} C_VEL
LIN {X 0,Y 28.792,Z 530.425,A -85,B 0,C 180,E1 -30822.922,E2 -30822.922} C_VEL
LIN {X 0,Y 21.616,Z 531.632,A -85,B 0,C 180,E1 -30851.029,E2 -30851.029} C_VEL
LIN {X 0,Y 20.618,Z 531.784,A -85,B 0,C 180,E1 -30870.002,E2 -30870.002} C_VEL
LIN {X 0,Y 24.516,Z 531.206,A -85,B 0,C 180,E1 -30904.986,E2 -30904.986} C_VEL
LIN {X 0,Y 33.899,Z 529.427,A -85,B 0,C 180,E1 -30926.028,E2 -30926.028} C_VEL
LIN {X 0,Y 45.655,Z 526.388,A -85,B 0,C 180,E1 -30937.464,E2 -30937.464} C_VEL
LIN {X 0,Y 58.482,Z 521.999,A -85,B 0,C 180,E1 -30944.03,E2 -30944.03} C_VEL
LIN {X 0,Y 68.397,Z 517.747,A -85,B 0,C 180,E1 -30947.468,E2 -30947.468} C_VEL
LIN {X 0,Y 78.47,Z 512.64,A -85,B 0,C 180,E1 -30950.134,E2 -30950.134} C_VEL
LIN {X 0,Y 88.691,Z 506.452,A -85,B 0,C 180,E1 -30952.112,E2 -30952.112} C_VEL
LIN {X 0,Y 91.38,Z 504.64,A -85,B 0,C 180,E1 -30953.596,E2 -30953.596} C_VEL
LIN {X 0,Y 91.827,Z 504.277,A -85,B 0,C 180,E1 -30955.61,E2 -30955.61} C_VEL
LIN {X 0,Y 91.694,Z 504.567,A -85,B 0,C 180,E1 -30960.351,E2 -30960.351} C_VEL
LIN {X 0,Y 90.622,Z 505.421,A -85,B 0,C 180,E1 -30961.446,E2 -30961.446} C_VEL
LIN {X 0,Y 88.854,Z 506.622,A -85,B 0,C 180,E1 -30962.04,E2 -30962.04} C_VEL
LIN {X 0,Y 85.006,Z 509.084,A -85,B 0,C 180,E1 -30962.186,E2 -30962.186} C_VEL
LIN {X 0,Y 76.176,Z 513.957,A -85,B 0,C 180,E1 -30960.967,E2 -30960.967} C_VEL
LIN {X 0,Y 73.382,Z 515.394,A -85,B 0,C 180,E1 -30961.094,E2 -30961.094} C_VEL
LIN {X 0,Y 59.853,Z 521.619,A -85,B 0,C 180,E1 -30963.532,E2 -30963.532} C_VEL
LIN {X 0,Y 46.091,Z 526.549,A -85,B 0,C 180,E1 -30967.628,E2 -30967.628} C_VEL
LIN {X 0,Y 36.024,Z 529.341,A -85,B 0,C 180,E1 -30972.715,E2 -30972.715} C_VEL
LIN {X 0,Y 23.393,Z 531.912,A -85,B 0,C 180,E1 -30985.668,E2 -30985.668} C_VEL
LIN {X 0,Y 14.112,Z 533.234,A -85,B 0,C 180,E1 -31020.127,E2 -31020.127} C_VEL
LIN {X 0,Y 13.032,Z 533.422,A -85,B 0,C 180,E1 -31049.997,E2 -31049.997} C_VEL
LIN {X 0,Y 17.985,Z 532.704,A -85,B 0,C 180,E1 -31101.4,E2 -31101.4} C_VEL
LIN {X 0,Y 29.522,Z 530.729,A -85,B 0,C 180,E1 -31122.219,E2 -31122.219} C_VEL
LIN {X 0,Y 42.686,Z 527.479,A -85,B 0,C 180,E1 -31131.062,E2 -31131.062} C_VEL
LIN {X 0,Y 56.386,Z 522.882,A -85,B 0,C 180,E1 -31135.655,E2 -31135.655} C_VEL
LIN {X 0,Y 70.305,Z 516.807,A -85,B 0,C 180,E1 -31138.459,E2 -31138.459} C_VEL
LIN {X 0,Y 81.676,Z 510.628,A -85,B 0,C 180,E1 -31140.138,E2 -31140.138} C_VEL
LIN {X 0,Y 84.338,Z 509.052,A -85,B 0,C 180,E1 -31140.436,E2 -31140.436} C_VEL
LIN {X 0,Y 85.758,Z 508.033,A -85,B 0,C 180,E1 -31142.855,E2 -31142.855} C_VEL
LIN {X 0,Y 84.523,Z 508.8,A -85,B 0,C 180,E1 -31143.808,E2 -31143.808} C_VEL
LIN {X 0,Y 73.152,Z 515.097,A -85,B 0,C 180,E1 -31145.514,E2 -31145.514} C_VEL
LIN {X 0,Y 60.368,Z 520.883,A -85,B 0,C 180,E1 -31148.284,E2 -31148.284} C_VEL
LIN {X 0,Y 46.779,Z 525.661,A -85,B 0,C 180,E1 -31152.436,E2 -31152.436} C_VEL
LIN {X 0,Y 36.883,Z 528.339,A -85,B 0,C 180,E1 -31157.685,E2 -31157.685} C_VEL
LIN {X 0,Y 24.511,Z 530.77,A -85,B 0,C 180,E1 -31170.666,E2 -31170.666} C_VEL
LIN {X 0,Y 15.082,Z 531.977,A -85,B 0,C 180,E1 -31202.229,E2 -31202.229} C_VEL
LIN {X 0,Y 13.526,Z 532.129,A -85,B 0,C 180,E1 -31230.003,E2 -31230.003} C_VEL
LIN {X 0,Y 19.131,Z 531.551,A -85,B 0,C 180,E1 -31277.286,E2 -31277.286} C_VEL
LIN {X 0,Y 30.51,Z 529.771,A -85,B 0,C 180,E1 -31297.137,E2 -31297.137} C_VEL
LIN {X 0,Y 43.427,Z 526.734,A -85,B 0,C 180,E1 -31306.176,E2 -31306.176} C_VEL
LIN {X 0,Y 56.941,Z 522.344,A -85,B 0,C 180,E1 -31310.908,E2 -31310.908} C_VEL
LIN {X 0,Y 67.212,Z 518.097,A -85,B 0,C 180,E1 -31313.408,E2 -31313.408} C_VEL
LIN {X 0,Y 79.625,Z 511.836,A -85,B 0,C 180,E1 -31315.623,E2 -31315.623} C_VEL
LIN {X 0,Y 84.515,Z 509.017,A -85,B 0,C 180,E1 -31316.284,E2 -31316.284} C_VEL
LIN {X 0,Y 85.816,Z 508.218,A -85,B 0,C 180,E1 -31317.435,E2 -31317.435} C_VEL
LIN {X 0,Y 85.803,Z 508.271,A -85,B 0,C 180,E1 -31318.519,E2 -31318.519} C_VEL
LIN {X 0,Y 84.34,Z 509.261,A -85,B 0,C 180,E1 -31319.597,E2 -31319.597} C_VEL
LIN {X 0,Y 73.382,Z 515.394,A -85,B 0,C 180,E1 -31321.094,E2 -31321.094} C_VEL
LIN {X 0,Y 67.214,Z 518.392,A -85,B 0,C 180,E1 -31321.55,E2 -31321.55} C_VEL
LIN {X 0,Y 56.593,Z 522.688,A -85,B 0,C 180,E1 -31320.701,E2 -31320.701} C_VEL
LIN {X 0,Y 47.91,Z 525.594,A -85,B 0,C 180,E1 -31319.626,E2 -31319.626} C_VEL
LIN {X 0,Y 41.304,Z 527.463,A -85,B 0,C 180,E1 -31319.663,E2 -31319.663} C_VEL
LIN {X 0,Y 39.105,Z 528.016,A -85,B 0,C 180,E1 -31320.079,E2 -31320.079} C_VEL
LIN {X 0,Y 28.176,Z 530.439,A -85,B 0,C 180,E1 -31323.835,E2 -31323.835} C_VEL
LIN {X 0,Y 14.636,Z 532.38,A -85,B 0,C 180,E1 -31336.167,E2 -31336.167} C_VEL
LIN {X 0,Y 5.907,Z 533.075,A -85,B 0,C 180,E1 -31409.993,E2 -31409.993} C_VEL
LIN {X 0,Y 14.626,Z 532.355,A -85,B 0,C 180,E1 -31483.942,E2 -31483.942} C_VEL
LIN {X 0,Y 28.17,Z 530.379,A -85,B 0,C 180,E1 -31496.298,E2 -31496.298} C_VEL
LIN {X 0,Y 42.171,Z 527.129,A -85,B 0,C 180,E1 -31500.744,E2 -31500.744} C_VEL
LIN {X 0,Y 49.225,Z 525.006,A -85,B 0,C 180,E1 -31501.994,E2 -31501.994} C_VEL
LIN {X 0,Y 49.265,Z 524.963,A -85,B 0,C 180,E1 -31503.032,E2 -31503.032} C_VEL
LIN {X 0,Y 35.378,Z 528.686,A -85,B 0,C 180,E1 -31506.651,E2 -31506.651} C_VEL
LIN {X 0,Y 21.766,Z 531.116,A -85,B 0,C 180,E1 -31514.386,E2 -31514.386} C_VEL
LIN {X 0,Y 9.414,Z 532.322,A -85,B 0,C 180,E1 -31541.716,E2 -31541.716} C_VEL
LIN {X 0,Y 6.452,Z 532.473,A -85,B 0,C 180,E1 -31590.006,E2 -31590.006} C_VEL
LIN {X 0,Y 15.239,Z 531.896,A -85,B 0,C 180,E1 -31657.284,E2 -31657.284} C_VEL
LIN {X 0,Y 28.509,Z 530.116,A -85,B 0,C 180,E1 -31670.433,E2 -31670.433} C_VEL
LIN {X 0,Y 42.295,Z 527.08,A -85,B 0,C 180,E1 -31675.581,E2 -31675.581} C_VEL
LIN {X 0,Y 49.264,Z 525.06,A -85,B 0,C 180,E1 -31677.024,E2 -31677.024} C_VEL
LIN {X 0,Y 49.226,Z 525.103,A -85,B 0,C 180,E1 -31678.035,E2 -31678.035} C_VEL
LIN {X 0,Y 39.105,Z 528.016,A -85,B 0,C 180,E1 -31680.079,E2 -31680.079} C_VEL
LIN {X 0,Y 37.6,Z 529.96,A -85,B 0,C 180,E1 -31680.481,E2 -31680.481} C_VEL
LIN {X 0,Y 37.6,Z 600,A -85,B 0,C 180,E1 -31680.481,E2 -31680.481} C_VEL
LIN {X 0,Y 37.6,Z 600,A -85,B 0,C 180,E1 -31680.481,E2 -31680.481}

QRS_NEXT_CUT()

QRS_NEXT()
QRS_HOME()

END
